Staubli VAL3: dateBase.pjx

--- dateBase.pjx ---
Parameters version=s7.3.1 stackSize=5000 millimeterUnit=true
Program file=start.pgx
Program file=stop.pgx
Data file=dateBase.dtx

--- dateBase.dtx ---
public bool bCenterPoint = true
public bool bFrameTeach = true
public bool bPLC
public bool bToolTeach
public bool bWorTbMoving
public frame fWorkTable = {x=1611.678918, y=32.649586, z=-207.483773, rx=4.556742, ry=-0.261146, rz=5.135586, fatherId=world[0]}
public jointRx jHome = {j1=40.634813, j2=24.616005, j3=104.715218, j4=-108.663007, j5=68.526435, j6=132.709111}
public mdesc mGrindingSpd = {accel=80, decel=70, tmax=100, leave=0.5, reach=0.5}
public mdesc mNomSpeed = {accel=36, vel=60, decel=36, rmax=2000, tmax=100, blend=cartesian, leave=5, reach=5}
public num nPrdRadius = 264.463067
public tool tTCP = {x=-12.113679, y=2.514779, z=192.872851, rx=33.798326, ry=31.269905, rz=-56.042932, fatherId=flange[0], ioLink=valve1}
